Fanuc KAREL source: kt00401.KL

-- PROVISIONAL review KL for V770-1; original PC SHA256 5c29aae8c0d4ba0d8ac0f54aaa59729de720fa16296a5b7a8cd0f6f26c55a2f0
-- Incomplete behavior may be omitted. Consult companion uncertainty JSON. Do not deploy.
PROGRAM KT00401
%NOLOCKGROUP
VAR
  I1 : INTEGER
  I2 : INTEGER
  OUT : BOOLEAN
BEGIN
  -- UNRESOLVED_PC offsets 5-16; opcodes 2E,23
  -- UNRESOLVED_PC offsets 21-32; opcodes 2E,23
  -- UNRESOLVED_PC offsets 37-48; opcodes 2E,23
  -- UNRESOLVED_PC offsets 53-64; opcodes 2E,23
  -- UNRESOLVED_PC offsets 69-88; opcodes 21,21,5B,23
  -- UNRESOLVED_PC offsets 93-97; opcodes 7F
END KT00401
